# EPICS IOC start-up script: iocsh/superv-common.iocsh
epicsEnvSet("D", "UCD-SNMP-MIB::")
epicsEnvSet("W", "SNMPv2-MIB::")
epicsEnvSet("N", "NOTIFICATION-LOG-MIB::")
epicsEnvSet("HR", "HOST-RESOURCES-MIB::")

# FREIA general status and NUC's ram disk usage
# dbLoadRecords("freia-status.db","HI=70,HH=90")

# Special records for getting Epics time since Epics epoch
#dbLoadRecords("epochTime.db")

# Scan server status
dbLoadRecords("scan.db","P=MJCtrl-scanserver:")
